// TIA Portal V21 export
DATA_BLOCK "RTC_to_String_Conversion Block"   // DB119
{ S7_Optimized_Access := 'TRUE' }
// stored: AutoNumber false, MemoryReserve 100
   VAR
      date_int : Int;
      date_string : String[6];
      month_int : Int;
      month_string : String[6];
      year_string : String[6];
      hour_int : Int;
      hour_string : String[6];
      minute_int : Int;
      minute_string : String[6];
      second_int : Int;
      second_string : String[6];
      date_temp : String[6];
      date_zero : Int;
      date_actual : String[12];
      month_temp : String[6];
      month_zero : Int;
      month_actual : String[6];
      year_actual : String[6];
      hour_temp : String[6];
      hour_zero : Int;
      hour_actual : String[6];
      minute_temp : String[6];
      minute_zero : Int;
      minute_actual : String[6];
      second_temp : String[6];
      second_zero : Int;
      second_actual : String[12];
      Final_Date : String[12];
      Final_time_HRS : String[12];
      Final_time_MINS : String[12];
      Final_time_1 : String[12];
      Final_time : String[8];
      SPACE : String[10];
   END_VAR
BEGIN
END_DATA_BLOCK
